FUNCTION F_SetAllMoversMovement : BOOL
VAR_INPUT
	Set			:ST_MoveDynamics;
END_VAR
VAR
	i			:UDINT;
END_VAR

FOR i:=1 TO XPlanar.MoverCount DO
	IF ip.Movers[i]<>0 THEN
		ip.Movers[i].Dynamics.Movement:=Set;		
	END_IF			
END_FOR

END_FUNCTION

(* stored: Version 1.1.0.1, ProductVersion 3.1.4026.18
   POU F_SetAllMoversMovement: Id {b1e646bf-97ca-48c6-8736-aa752c85bfcf}, SpecialFunc None *)
